// TIA Portal V20 export
// export: Created 2026-04-11T06:02:30.695832Z, ExportSetting WithDefaults, DisplayName Totally Integrated Automation Portal, DisplayVersion V20, DisplayName TIA Portal Openness, DisplayVersion V20, DisplayName TIA Portal Version Control Interface, DisplayVersion V20, DisplayName STEP 7 Professional, DisplayVersion V20, DisplayName STEP 7 Safety, DisplayVersion V20, DisplayName WinCC Basic/Comfort/Advanced, DisplayVersion V20, DisplayName WinCC Unified, DisplayVersion V20
TYPE "udtHMI_PID"
// stored: IsFailsafeCompliant false
   STRUCT
      iPIDMode : Int;   // Current Mode of the PID block
      rProcessValue { ExternalWritable := 'False'} : Real;   // Current Process Value
      rOutput { ExternalWritable := 'False'} : Real;   // Current Output
      rAutoOutput { ExternalWritable := 'False'} : Real;   // Auto mode output
      rManualOutput { S7_SetPoint := 'True'} : Real;   // Manual mode output
      rOutputIntegral { ExternalWritable := 'False'} : Real;   // The integral component of the current CV
      rOutputProportional { ExternalWritable := 'False'} : Real;   // The proportional component of the current CV
      rOutputDerivative { ExternalWritable := 'False'} : Real;   // The derivative component of the current CV
      rAutoSP { ExternalWritable := 'False'} : Real;   // Auto mode setpoint
      rManualSP { S7_SetPoint := 'True'} : Real;   // Manual mode setpoint
      bPB_OverrideSP : Bool;   // PB Override automatic mode setpoint
      bTOG_OverrideSP { ExternalWritable := 'False'} : Bool;   // Auto mode setpoint overriden
      bPB_Reset : Bool;   // PB Reset integral wind up
      bPBEN_OverrideSP { ExternalWritable := 'False'} : Bool;   // PB Override auto mode setpoint enabled
      bPBEN_Reset : Bool;   // PB Reset integral wind up enabled
      bShowTuningPage : Bool;   // PB to showing tuning page
      Config : "udtHMI_PID_Config";
   END_STRUCT;
END_TYPE
